# EPICS autosave request: CARSApp/Db/CARS_54_motor_positions.req
# FILE... CARS_56_motor_settings.req
file "motor_positions.req", P=$(P), M=m1
file "motor_positions.req", P=$(P), M=m2
file "motor_positions.req", P=$(P), M=m3
file "motor_positions.req", P=$(P), M=m4
file "motor_positions.req", P=$(P), M=m5
file "motor_positions.req", P=$(P), M=m6
file "motor_positions.req", P=$(P), M=m7
file "motor_positions.req", P=$(P), M=m8
file "motor_positions.req", P=$(P), M=m9
file "motor_positions.req", P=$(P), M=m10
file "motor_positions.req", P=$(P), M=m11
file "motor_positions.req", P=$(P), M=m12
file "motor_positions.req", P=$(P), M=m13
file "motor_positions.req", P=$(P), M=m14
file "motor_positions.req", P=$(P), M=m15
file "motor_positions.req", P=$(P), M=m16
file "motor_positions.req", P=$(P), M=m17
file "motor_positions.req", P=$(P), M=m18
file "motor_positions.req", P=$(P), M=m19
file "motor_positions.req", P=$(P), M=m20
file "motor_positions.req", P=$(P), M=m21
file "motor_positions.req", P=$(P), M=m22
file "motor_positions.req", P=$(P), M=m23
file "motor_positions.req", P=$(P), M=m24
file "motor_positions.req", P=$(P), M=m25
file "motor_positions.req", P=$(P), M=m26
file "motor_positions.req", P=$(P), M=m27
file "motor_positions.req", P=$(P), M=m28
file "motor_positions.req", P=$(P), M=m29
file "motor_positions.req", P=$(P), M=m30
file "motor_positions.req", P=$(P), M=m31
file "motor_positions.req", P=$(P), M=m32
file "motor_positions.req", P=$(P), M=m33
file "motor_positions.req", P=$(P), M=m34
file "motor_positions.req", P=$(P), M=m35
file "motor_positions.req", P=$(P), M=m36
file "motor_positions.req", P=$(P), M=m37
file "motor_positions.req", P=$(P), M=m38
file "motor_positions.req", P=$(P), M=m39
file "motor_positions.req", P=$(P), M=m40
file "motor_positions.req", P=$(P), M=m41
file "motor_positions.req", P=$(P), M=m42
file "motor_positions.req", P=$(P), M=m43
file "motor_positions.req", P=$(P), M=m44
file "motor_positions.req", P=$(P), M=m45
file "motor_positions.req", P=$(P), M=m46
file "motor_positions.req", P=$(P), M=m47
file "motor_positions.req", P=$(P), M=m48
file "motor_positions.req", P=$(P), M=m49
file "motor_positions.req", P=$(P), M=m50
file "motor_positions.req", P=$(P), M=m51
file "motor_positions.req", P=$(P), M=m52
file "motor_positions.req", P=$(P), M=m53
file "motor_positions.req", P=$(P), M=m54
